// TwinCAT 3 PLC project SerialCommunication
// Title: SerialCom_Lib
// Company: Chua Siang Poh
// Author: Chua Siang Poh
// ProjectVersion: 2.0.1
// Description: Device library designed for simpler and modular serial communication applications in TwinCAT. Number of serial com channels can be specified in the Parameter list.
// ProgramVersion: 3.1.4020.10
// libraries:
//   Tc2_SerialCom, * (Beckhoff Automation GmbH)
//   Tc2_Standard, * (Beckhoff Automation GmbH)
//   Tc2_System, * (Beckhoff Automation GmbH)
//   Tc3_Interfaces, * (Beckhoff Automation GmbH)
//   Tc3_Module, * (Beckhoff Automation GmbH)
// project tree:
//   Base Component/Class/Common Base/ C_SERIALCOMM_PORT.TcPOU
//   Base Component/Class/ C_SERIALCOMM_EL6.TcPOU, C_SERIALCOMM_PC.TcPOU
//   Base Component/Interfaces/ I_SERIALCONTROLLER.TcIO (not stored)
//   Version/ Global_Version.TcGVL

// ---- Version/Global_Version.TcGVL
{attribute 'TcGenerated'}
// This function has been automatically generated from the project information.
VAR_GLOBAL CONSTANT
	{attribute 'const_non_replaced'}
	{attribute 'linkalways'}
	stLibVersion_SerialCom_Lib : ST_LibVersion := (iMajor := 2, iMinor := 0, iBuild := 1, iRevision := 0, sVersion := '2.0.1');
END_VAR

// ---- Base Component/Class/Common Base/C_SERIALCOMM_PORT.TcPOU
FUNCTION_BLOCK C_SERIALCOMM_PORT IMPLEMENTS I_SERIALCONTROLLER
VAR_INPUT
END_VAR
VAR_OUTPUT
END_VAR
VAR
	//Software Buffer
		_txbuffer 		: ComBuffer;
		_rxbuffer		: ComBuffer;	
	//Internal Memory Buffer
		_buffer 	: ARRAY[0..3000] OF BYTE;
	C_LINECONTROL 	: SerialLineControl;
	C_SendData 		: SendData;
	C_ReceiveData	: ReceiveData;
	_prefix, _suffix: STRING(15);
	_timeout 		: TIME := T#500MS;
END_VAR

METHOD UPDATE_BUFFER : DINT
{warning 'Hardware function is not implemented in Serial Comm base class'}
UPDATE_BUFFER := 0;
RETURN;
END_METHOD

PROPERTY RECEIVE_PREFIX : STRING(15)
SET
_prefix := prefix;
END_SET
GET
Prefix := _prefix;
END_GET
END_PROPERTY

METHOD SEND : DINT
VAR_INPUT
	ptr_data 	: PVOID;
	length		: UDINT;
END_VAR
C_SendData(
	pSendData:= ptr_data, 
	Length:= length, 
	TXbuffer:= _txbuffer);
IF C_SendData.Error <> COMERROR_NOERROR THEN
	Send := 1;
	RETURN;
ELSIF NOT C_SendData.Busy THEN
	Send := -1;
	RETURN;
ELSE
	Send := 0;
	RETURN;
END_IF
END_METHOD

METHOD RECEIVE : DINT
VAR_INPUT
	ptr_data 	: PVOID;
END_VAR
VAR
END_VAR
IF LEN(_prefix) > 0 THEN
	C_ReceiveData.pPrefix := ADR(_prefix);
	C_ReceiveData.LenPrefix := INT_TO_BYTE(LEN(_prefix));
ELSE
	C_ReceiveData.pPrefix := 0;
	C_ReceiveData.LenPrefix := 0;
END_IF
IF LEN(_suffix) > 0 THEN
	C_ReceiveData.pSuffix := ADR(_suffix);
	C_ReceiveData.LenSuffix := INT_TO_BYTE(LEN(_suffix));
ELSE
	C_ReceiveData.pSuffix := 0;
	C_ReceiveData.LenSuffix := 0;
END_IF
C_ReceiveData(
	pReceiveData:= ADR(_buffer), 
	SizeReceiveData:= SIZEOF(_buffer), 
	Timeout:= _timeout, 
	LenReceiveData=> , 
	RXbuffer:= _rxbuffer);
IF C_ReceiveData.Error <> COMERROR_NOERROR THEN
	Receive := 1;
	RETURN;
ELSIF C_ReceiveData.DataReceived THEN
	MEMCPY(ptr_data, ADR(_buffer), C_ReceiveData.LenReceiveData);
	Receive := -1;
	RETURN;
ELSE
	Receive := 0;
	RETURN;
END_IF
END_METHOD

PROPERTY TIMEOUT : TIME
GET
TimeOut := _timeout;
END_GET
SET
_timeout := timeout;
END_SET
END_PROPERTY

PROPERTY RECEIVE_SUFFIX : STRING(15)
GET
RECEIVE_SUFFIX := _suffix;
END_GET
SET
_suffix := RECEIVE_SUFFIX;
END_SET
END_PROPERTY

END_FUNCTION_BLOCK

// ---- Base Component/Class/C_SERIALCOMM_EL6.TcPOU
FUNCTION_BLOCK C_SERIALCOMM_EL6 EXTENDS C_SERIALCOMM_PORT
VAR_INPUT
END_VAR
VAR_OUTPUT
END_VAR
VAR
	_hwRxBuffer		AT %I* : EL6inData22B;
	_hwTxBuffer		AT %Q* : EL6outData22B;
END_VAR

METHOD UPDATE_BUFFER : DINT
{message 'PC type Comm Port implemented'}
C_LINECONTROL(
	Mode:= SERIALLINEMODE_EL6_22B, 
	pComIn:= ADR(_hwRxBuffer), 
	pComOut:= ADR(_hwTxBuffer), 
	SizeComIn:= SIZEOF(_hwRxBuffer), 
	TxBuffer:= _txbuffer, 
	RxBuffer:= _rxbuffer);
	
IF C_LINECONTROL.Error THEN
	UPDATE_BUFFER := 1;
	RETURN;
ELSE
	UPDATE_BUFFER := -1;
	RETURN;
END_IF
END_METHOD

END_FUNCTION_BLOCK

// ---- Base Component/Class/C_SERIALCOMM_PC.TcPOU
FUNCTION_BLOCK C_SERIALCOMM_PC EXTENDS C_SERIALCOMM_PORT
VAR_INPUT
END_VAR
VAR_OUTPUT
END_VAR
VAR
	_hwRxBuffer		AT %I* : PcComInData;
	_hwTxBuffer		AT %Q* : PcComOutData;
END_VAR

METHOD UPDATE_BUFFER : DINT
{message 'PC type Comm Port implemented'}
C_LINECONTROL(
	Mode:= SERIALLINEMODE_PC_COM_PORT, 
	pComIn:= ADR(_hwRxBuffer), 
	pComOut:= ADR(_hwTxBuffer), 
	SizeComIn:= SIZEOF(_hwRxBuffer), 
	TxBuffer:= _txbuffer, 
	RxBuffer:= _rxbuffer);
		
IF C_LINECONTROL.Error THEN
	UPDATE_BUFFER := 1;
	RETURN;
ELSE
	UPDATE_BUFFER := -1;
	RETURN;
END_IF
END_METHOD

END_FUNCTION_BLOCK
